FUNCTION_BLOCK Overcurrent_Protector (* Extracted Composite Function Block Type *)
  (* Standard: 61499-2 *)
  (* Version 1/31/2024, Maxth *)
  PACKAGE Main;
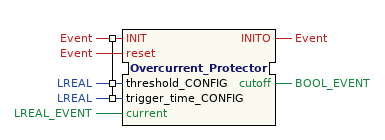
  EVENT_INPUT
    INIT WITH threshold_CONFIG, trigger_time_CONFIG;
    reset;
  END_EVENT
  EVENT_OUTPUT
    INITO;
  END_EVENT
  VAR_INPUT
    threshold_CONFIG : LREAL;
    trigger_time_CONFIG : LREAL;
  END_VAR
  SOCKETS
    current : LREAL_EVENT;
  END_SOCKETS
  PLUGS
    cutoff : BOOL_EVENT;
  END_PLUGS
  FBS
    FB1 : Current_Transformer(manual_currentMeasurement := 8);
    FB2 : Comparator(overcurrentThreshold := 10.0);
    FB7 : Circuit_Breaker;
  END_FBS
  EVENT_CONNECTIONS
    FB1.INITO TO FB2.INIT;
    FB1.AMPSV TO FB2.SAMPLE;
    INIT TO FB1.INIT;
    FB7.INITO TO INITO;
    FB2.OP TO FB7.OPOPN;
    FB2.INITO TO FB7.INIT;
  END_CONNECTIONS
  DATA_CONNECTIONS
    FB1.current_out TO FB2.AmpSV;
    FB2.Op TO FB7.OpOpn;
  END_CONNECTIONS
  ADAPTER_CONNECTIONS
    current TO FB1.current_in;
    FB7.GOOSE TO cutoff;
  END_CONNECTIONS
END_FUNCTION_BLOCK
